Returns 0.0 for unsupported types — caller must verify TypeClass first.
Mirrors the dispatch in FB_TcOtelTaskTracer.AddAny so trace and metric
emission see numerics consistently.
*)
METHOD PRIVATE _AnyToLreal : LREAL
VAR_INPUT
    stArg : ANY;
END_VAR
VAR
    pBool  : POINTER TO BYTE;
    pSint  : POINTER TO SINT;
    pInt   : POINTER TO INT;
    pDint  : POINTER TO DINT;
    pLint  : POINTER TO LINT;
    pUsint : POINTER TO USINT;
    pUint  : POINTER TO UINT;
    pUdint : POINTER TO UDINT;
    pUlint : POINTER TO ULINT;
    pReal  : POINTER TO REAL;
    pLreal : POINTER TO LREAL;
END_VAR
CASE stArg.TypeClass OF
    __SYSTEM.TYPE_CLASS.TYPE_BOOL:
        pBool := stArg.pValue;
        IF pBool^ <> 0 THEN
            _AnyToLreal := 1.0;
        ELSE
            _AnyToLreal := 0.0;
        END_IF

    __SYSTEM.TYPE_CLASS.TYPE_SINT:
        pSint := stArg.pValue;
        _AnyToLreal := SINT_TO_LREAL(pSint^);

    __SYSTEM.TYPE_CLASS.TYPE_INT:
        pInt := stArg.pValue;
        _AnyToLreal := INT_TO_LREAL(pInt^);

    __SYSTEM.TYPE_CLASS.TYPE_DINT:
        pDint := stArg.pValue;
        _AnyToLreal := DINT_TO_LREAL(pDint^);

    __SYSTEM.TYPE_CLASS.TYPE_LINT:
        pLint := stArg.pValue;
        _AnyToLreal := LINT_TO_LREAL(pLint^);

    __SYSTEM.TYPE_CLASS.TYPE_USINT,
    __SYSTEM.TYPE_CLASS.TYPE_BYTE:
        pUsint := stArg.pValue;
        _AnyToLreal := USINT_TO_LREAL(pUsint^);

    __SYSTEM.TYPE_CLASS.TYPE_UINT,
    __SYSTEM.TYPE_CLASS.TYPE_WORD:
        pUint := stArg.pValue;
        _AnyToLreal := UINT_TO_LREAL(pUint^);

    __SYSTEM.TYPE_CLASS.TYPE_UDINT,
    __SYSTEM.TYPE_CLASS.TYPE_DWORD:
        pUdint := stArg.pValue;
        _AnyToLreal := UDINT_TO_LREAL(pUdint^);

    __SYSTEM.TYPE_CLASS.TYPE_ULINT,
    __SYSTEM.TYPE_CLASS.TYPE_LWORD:
        pUlint := stArg.pValue;
        _AnyToLreal := ULINT_TO_LREAL(pUlint^);

    __SYSTEM.TYPE_CLASS.TYPE_REAL:
        pReal := stArg.pValue;
        _AnyToLreal := REAL_TO_LREAL(pReal^);

    __SYSTEM.TYPE_CLASS.TYPE_LREAL:
        pLreal := stArg.pValue;
        _AnyToLreal := pLreal^;

    ELSE
        _AnyToLreal := 0.0;
END_CASE
END_METHOD

(*
:Description: Snapshot the current Welford aggregator into the body buffer.

Writes ``popcount(_nStatMask) * 8`` bytes — one LREAL per set bit, in
bit-index order (Min, Max, Mean, Sum, Count, StdDev). Returns FALSE on
body overflow without touching the buffer; the caller marks ``_bOverflow``.

Empty windows (no Observe call landed since the previous snapshot) still
produce a sample slot — all zeros — so ``sample_count`` keeps matching the
expected wall-clock cadence on the receiver side.
*)
METHOD PRIVATE _AppendAggregated : BOOL
VAR_INPUT
    (* Cycle offset for this sample relative to _nCycleStart. Only written
       when _bRecordSampleTimes is TRUE; ignored otherwise. Callers pass 0
       when they don't care. *)
    nCycleOff : UINT;
    (* Absolute DC time for this sample (raw F_GetActualDcTime64). Only
       written when _bRecordSampleTimesDc is TRUE; ignored otherwise. *)
    nDcSample : LINT;
END_VAR
VAR
    pDst    : POINTER TO BYTE;
    nOffset : UDINT;
    nStride : UDINT;
    fStdDev : LREAL;
    fCount  : LREAL;
END_VAR
nStride := _nSampleSize;
IF _bRecordSampleTimes THEN
    nStride := nStride + 2;
ELSIF _bRecordSampleTimesDc THEN
    nStride := nStride + 8;
END_IF
IF (_nBodyOffset + nStride) > BODY_CAPACITY THEN
    _AppendAggregated := FALSE;
    RETURN;
END_IF

pDst    := _ActiveBodyPtr() + _nBodyOffset;
IF _bRecordSampleTimes THEN
    Tc2_System.MEMCPY(pDst, ADR(nCycleOff), 2);
    pDst := pDst + 2;
ELSIF _bRecordSampleTimesDc THEN
    Tc2_System.MEMCPY(pDst, ADR(nDcSample), 8);
    pDst := pDst + 8;
END_IF
nOffset := 0;

IF (_nStatMask AND E_MetricStat.eMin) <> 0 THEN
    Tc2_System.MEMCPY(pDst + nOffset, ADR(_aggMin), 8);
    nOffset := nOffset + 8;
END_IF
IF (_nStatMask AND E_MetricStat.eMax) <> 0 THEN
    Tc2_System.MEMCPY(pDst + nOffset, ADR(_aggMax), 8);
    nOffset := nOffset + 8;
END_IF
IF (_nStatMask AND E_MetricStat.eMean) <> 0 THEN
    Tc2_System.MEMCPY(pDst + nOffset, ADR(_aggMean), 8);
    nOffset := nOffset + 8;
END_IF
IF (_nStatMask AND E_MetricStat.eSum) <> 0 THEN
    Tc2_System.MEMCPY(pDst + nOffset, ADR(_aggSum), 8);
    nOffset := nOffset + 8;
END_IF
IF (_nStatMask AND E_MetricStat.eCount) <> 0 THEN
    fCount := UDINT_TO_LREAL(_nAggCount);
    Tc2_System.MEMCPY(pDst + nOffset, ADR(fCount), 8);
    nOffset := nOffset + 8;
END_IF
IF (_nStatMask AND E_MetricStat.eStdDev) <> 0 THEN
    IF _nAggCount > 1 THEN
        fStdDev := SQRT(_aggSumSq / UDINT_TO_LREAL(_nAggCount - 1));
    ELSE
        fStdDev := 0.0;
    END_IF
    Tc2_System.MEMCPY(pDst + nOffset, ADR(fStdDev), 8);
    nOffset := nOffset + 8;
END_IF

_nBodyOffset      := _nBodyOffset + nStride;
_nSampleCount     := _nSampleCount + 1;
_AppendAggregated := TRUE;
END_METHOD

(*
:Description: Write one sample of the locked schema into the body buffer.

Returns FALSE when the body is full — caller sets ``_bOverflow``.
*)
METHOD PRIVATE _AppendSample : BOOL
VAR_INPUT
    stArg     : ANY;
    (* Cycle offset for this sample relative to _nCycleStart. Only written
       when _bRecordSampleTimes is TRUE; ignored otherwise. Callers pass 0
       when they don't care. *)
    nCycleOff : UINT;
    (* Absolute DC time for this sample (raw F_GetActualDcTime64). Only
       written when _bRecordSampleTimesDc is TRUE; ignored otherwise. *)
    nDcSample : LINT;
END_VAR
VAR
    fLreal     : LREAL;
    nStrLen    : UDINT;
    nCopyLen   : UDINT;
    nStride    : UDINT;
    pDst       : POINTER TO BYTE;
    pWstr      : POINTER TO WSTRING(255);
END_VAR
nStride := _nSampleSize;
IF _bRecordSampleTimes THEN
    nStride := nStride + 2;
ELSIF _bRecordSampleTimesDc THEN
    nStride := nStride + 8;
END_IF
IF (_nBodyOffset + nStride) > BODY_CAPACITY THEN
    _AppendSample := FALSE;
    RETURN;
END_IF

pDst := _ActiveBodyPtr() + _nBodyOffset;
IF _bRecordSampleTimes THEN
    Tc2_System.MEMCPY(pDst, ADR(nCycleOff), 2);
    pDst := pDst + 2;
ELSIF _bRecordSampleTimesDc THEN
    Tc2_System.MEMCPY(pDst, ADR(nDcSample), 8);
    pDst := pDst + 8;
END_IF

CASE _eBodySchema OF
    E_MetricBodySchema.eBool:
        IF Tc2_Utilities.PBYTE_TO_BYTE(stArg.pValue) <> 0 THEN
            pDst^ := 1;
        ELSE
            pDst^ := 0;
        END_IF

    E_MetricBodySchema.eNumeric:
        fLreal := _AnyToLreal(stArg);
        Tc2_System.MEMCPY(pDst, ADR(fLreal), 8);

    E_MetricBodySchema.eDiscrete:
        nCopyLen := DINT_TO_UDINT(stArg.diSize);
        IF nCopyLen > _nSampleSize THEN
            nCopyLen := _nSampleSize;
        END_IF
        Tc2_System.MEMCPY(pDst, stArg.pValue, nCopyLen);
        IF nCopyLen < _nSampleSize THEN
            Tc2_System.MEMSET(pDst + nCopyLen, 0, _nSampleSize - nCopyLen);
        END_IF

    E_MetricBodySchema.eString:
        Tc2_System.MEMSET(pDst, 0, _nSampleSize);
        nStrLen := Tc2_Utilities.LEN2(stArg.pValue);
        IF nStrLen > _nSampleSize THEN
            nStrLen := _nSampleSize;
        END_IF
        IF nStrLen > 0 THEN
            Tc2_System.MEMCPY(pDst, stArg.pValue, nStrLen);
        END_IF

    E_MetricBodySchema.eWstring:
        Tc2_System.MEMSET(pDst, 0, _nSampleSize);
        (* WLEN returns characters; we ship 2 B each, capped at _nSampleSize bytes.
           Typed-pointer cast first because WLEN can't take PVOID directly —
           same pattern FB_LogEntry._WriteWString uses. *)
        pWstr := stArg.pValue;
        nStrLen := INT_TO_UDINT(Tc2_Standard.WLEN(pWstr^)) * 2;
        IF nStrLen > _nSampleSize THEN
            nStrLen := _nSampleSize;
        END_IF
        IF nStrLen > 0 THEN
            Tc2_System.MEMCPY(pDst, stArg.pValue, nStrLen);
        END_IF

    ELSE
        _AppendSample := FALSE;
        RETURN;
END_CASE

_nBodyOffset  := _nBodyOffset + nStride;
_nSampleCount := _nSampleCount + 1;

_AppendSample := TRUE;
END_METHOD

(*
:Description: Flush if push window has elapsed.

Window timing is cycle-based (mirrors ``FB_TcOtelTaskDiag.CheckFlush``):
``target_cycles = push_interval_ms * 1000 / cycle_time_us``. Doesn't fire
when the buffer is empty — empty windows just slide the start cycle
forward.
*)
METHOD PRIVATE _CheckFlush
VAR
    nTaskIdx       : DINT;
    pTi            : POINTER TO PlcTaskSystemInfo;
    nNowCycle      : UDINT;
    nCycleTimeUs   : UDINT;
    nTargetCycles  : UDINT;
END_VAR
nTaskIdx := Tc2_Utilities.GETCURTASKINDEXEX();
IF nTaskIdx <= 0 THEN
    RETURN;
END_IF
pTi := ADR(TwinCAT_SystemInfoVarList._TaskInfo[nTaskIdx]);

nCycleTimeUs := pTi^.CycleTime / 10;
IF nCycleTimeUs = 0 THEN
    nCycleTimeUs := 1000; (* fallback: assume 1 ms *)
END_IF
nTargetCycles := (_nPushIntervalMs * 1000) / nCycleTimeUs;
IF nTargetCycles = 0 THEN
    nTargetCycles := 1;
END_IF

(* When per-sample timestamps are active, cap the window at the u16 ceiling
   so the per-sample cycle-offset never overflows. Observable effect: an
   earlier autoflush for extreme configs (e.g. 20 s push window on a 250 µs
   task). WithSpan pins may be consumed by the autoflush rather than the
   natural flush — use BindTracer for spans that outlive one window. *)
IF _bRecordSampleTimes AND nTargetCycles > 16#FFFF THEN
    nTargetCycles := 16#FFFF;
END_IF

nNowCycle := pTi^.CycleCount;
IF NOT _bWindowStartSet OR nNowCycle < _nWindowStartCycle THEN
    _nWindowStartCycle := nNowCycle;
    _bWindowStartSet   := TRUE;
    RETURN;
END_IF

IF (nNowCycle - _nWindowStartCycle) < nTargetCycles THEN
    RETURN;
END_IF

IF _nSampleCount > 0 THEN
    _DoFlush();
END_IF
_nWindowStartCycle := nNowCycle;
END_METHOD

(*
:Description: Finalize the active window into a sendable frame and enqueue for the sender.

Phase 8 — zero-copy queued dispatch:

1. If the previous window is still queued (``_bPending``) the sender has
   fallen behind. Increment ``_nDropWindow`` and reset the active half —
   we cannot touch the pending half nor duplicate ourselves in the queue.
2. Otherwise: build the header into a small stack staging (≤ ~160 B),
   MEMCPY the staged header into the active frame's reserve region so it
   sits directly before the body (one contiguous byte run), snapshot the
   pending metadata (buf index, hdr len, body len), flip ``_eActiveBuf``,
   reset the now-active (previously empty) half, and call
   ``sender.Enqueue(THIS)``.

The sender later calls ``_GetPendingPtr`` / ``_GetPendingLen`` to read the
frame pointer + length directly into ADSWRITE, and ``_NotifyFrameSent``
when the transfer completes. The body buffer is never MEMCPY'd.
*)
METHOD PRIVATE _DoFlush
VAR
    stHeader    : ST_PushMetricAggHeader;
    abyHdr      : ARRAY[0..255] OF BYTE;   // header(52) + trace(24) + name(63) + unit(15) + ns_len(1) + ns(127) ≤ 282
    nHdrLen     : UDINT;
    nNameLen    : UDINT;
    nUnitLen    : UDINT;
    nNsLen      : UDINT;
    byNsLen     : BYTE;
    refSender   : REFERENCE TO FB_TcOtelTaskMetrics;
    refSpan     : REFERENCE TO FB_Span;
    pActiveBase : POINTER TO BYTE;
END_VAR
(* Backlog guard: if the sender is still shipping our previous frame, the
   pending half is in use and we have no clean buffer to swap into. Drop
   this window rather than risk body corruption. In practice this only
   fires during a dead / slow tc-otel endpoint. *)
IF _bPending THEN
    _nDropWindow      := _nDropWindow + 1;
    _nBodyOffset      := 0;
    _nSampleCount     := 0;
    _bOverflow        := FALSE;
    _bWindowHasSample := FALSE;
    _nCycleStart      := 0;
    _nCycleEnd        := 0;
    _nDcTimeStart     := 0;
    _nDcTimeEnd       := 0;
    RETURN;
END_IF

(* Resolve trace context: per-flush WithSpan override beats persistent
   BindTracer. Both candidates and the chosen handle stay as REFERENCE TO —
   nullable via REF= 0 + __ISVALIDREF, no pointer round-trip needed. *)
refSpan REF= 0;
IF __ISVALIDREF(_pSpanOverride) THEN
    refSpan REF= _pSpanOverride;
ELSIF __ISVALIDREF(_pTracer) THEN
    refSpan REF= _pTracer.InnermostSpan;
END_IF

(* Build fixed header. *)
stHeader.nVersion         := 2;
stHeader.nEventType       := 21;
stHeader.nFlags           := 0;
IF _bOverflow THEN
    stHeader.nFlags := stHeader.nFlags OR 16#02;    (* bit1 = ring_overflowed *)
END_IF
IF __ISVALIDREF(refSpan) THEN
    stHeader.nFlags := stHeader.nFlags OR 16#01;    (* bit0 = has_trace_ctx *)
END_IF
IF _bRecordSampleTimes THEN
    stHeader.nFlags := stHeader.nFlags OR 16#04;    (* bit2 = has_sample_ts *)
END_IF
IF _bRecordSampleTimesDc THEN
    stHeader.nFlags := stHeader.nFlags OR 16#10;    (* bit4 = has_sample_ts_dc *)
END_IF
nNsLen := Tc2_Utilities.LEN2(ADR(_sLogger));
IF nNsLen > 127 THEN
    nNsLen := 127;
END_IF
IF nNsLen > 0 THEN
    stHeader.nFlags := stHeader.nFlags OR 16#08;    (* bit3 = has_namespace *)
END_IF
stHeader.eBodySchema      := _eBodySchema;
stHeader.nSampleSize      := _nSampleSize;
stHeader.nSampleCount     := _nSampleCount;
stHeader.nMetricId        := _nMetricId;
stHeader.nTaskIndex       := TO_USINT(Tc2_Utilities.GETCURTASKINDEXEX());
stHeader.nStatMask        := _nStatMask;
stHeader.nCycleCountStart := _nCycleStart;
stHeader.nCycleCountEnd   := _nCycleEnd;
stHeader.nDcTimeStart     := _nDcTimeStart;
stHeader.nDcTimeEnd       := _nDcTimeEnd;

nNameLen := Tc2_Utilities.LEN2(ADR(_sName));
IF nNameLen > 63 THEN
    nNameLen := 63;
END_IF
nUnitLen := Tc2_Utilities.LEN2(ADR(_sUnit));
IF nUnitLen > 15 THEN
    nUnitLen := 15;
END_IF
stHeader.nNameLen := TO_BYTE(nNameLen);
stHeader.nUnitLen := TO_BYTE(nUnitLen);

(* Stage [header | (trace_ctx) | name | unit] on the stack. *)
Tc2_System.MEMCPY(ADR(abyHdr), ADR(stHeader), SIZEOF(stHeader));
nHdrLen := SIZEOF(stHeader);

IF __ISVALIDREF(refSpan) THEN
    Tc2_System.MEMCPY(ADR(abyHdr) + nHdrLen,      ADR(refSpan._abTraceId[0]), 16);
    Tc2_System.MEMCPY(ADR(abyHdr) + nHdrLen + 16, ADR(refSpan._abSpanId[0]),  8);
    nHdrLen := nHdrLen + 24;
END_IF

(* Consume per-flush span override — BindTracer stays, WithSpan is one-shot. *)
_pSpanOverride REF= 0;

IF nNameLen > 0 THEN
    Tc2_System.MEMCPY(ADR(abyHdr) + nHdrLen, ADR(_sName), nNameLen);
    nHdrLen := nHdrLen + nNameLen;
END_IF
IF nUnitLen > 0 THEN
    Tc2_System.MEMCPY(ADR(abyHdr) + nHdrLen, ADR(_sUnit), nUnitLen);
    nHdrLen := nHdrLen + nUnitLen;
END_IF
IF nNsLen > 0 THEN
    (* Phase 2 scope-resolver: ns_len(1) + namespace(ns_len). *)
    byNsLen := TO_BYTE(nNsLen);
    Tc2_System.MEMCPY(ADR(abyHdr) + nHdrLen,     ADR(byNsLen),   1);
    Tc2_System.MEMCPY(ADR(abyHdr) + nHdrLen + 1, ADR(_sLogger),  nNsLen);
    nHdrLen := nHdrLen + 1 + nNsLen;
END_IF

(* Defensive clamp: the header reserve is HDR_RESERVE bytes. Oversized
   headers would overlap the body. In practice nHdrLen ≤ 154. *)
IF nHdrLen > HDR_RESERVE THEN
    _nDropEmit := _nDropEmit + 1;
    (* Reset window and bail — don't corrupt the frame layout. *)
    _nBodyOffset      := 0;
    _nSampleCount     := 0;
    _bOverflow        := FALSE;
    _bWindowHasSample := FALSE;
    _nCycleStart      := 0;
    _nCycleEnd        := 0;
    _nDcTimeStart     := 0;
    _nDcTimeEnd       := 0;
    RETURN;
END_IF

(* Position the staged header so its last byte sits at offset HDR_RESERVE-1
   of the active frame — i.e. flush against the body start. Single MEMCPY
   of ≤ 160 B; no body copy. *)
pActiveBase := _ActiveFrameAddr();
Tc2_System.MEMCPY(pActiveBase + (HDR_RESERVE - nHdrLen), ADR(abyHdr), nHdrLen);

(* Snapshot pending metadata: the active (now-to-be-shipped) half. *)
_ePendingBuf     := _eActiveBuf;
_nPendingHdrLen  := nHdrLen;
_nPendingBodyLen := _nBodyOffset;
_bPending        := TRUE;

(* Flip active → the other half. Reset the new-active mutable state. *)
IF _eActiveBuf = 0 THEN
    _eActiveBuf := 1;
ELSE
    _eActiveBuf := 0;
END_IF
_nBodyOffset      := 0;
_nSampleCount     := 0;
_bOverflow        := FALSE;
_bWindowHasSample := FALSE;
_nCycleStart      := 0;
_nCycleEnd        := 0;
_nDcTimeStart     := 0;
_nDcTimeEnd       := 0;

(* Hand the pending half to the sender's dispatch ring. *)
refSender REF= PRG_TaskLog.TaskMetrics;
IF __ISVALIDREF(refSender) THEN
    IF NOT refSender.Enqueue(THIS) THEN
        (* Ring overflow — real drop. Release the pending half so the next
           window can still flush, and count as emit drop. *)
        _bPending  := FALSE;
        _nDropEmit := _nDropEmit + 1;
    END_IF
ELSE
    (* Sender missing — treat like ring overflow. *)
    _bPending  := FALSE;
    _nDropEmit := _nDropEmit + 1;
END_IF
END_METHOD

(*
:Description: INTERNAL — total bytes of the frame currently in the sender queue.

Called by ``FB_TcOtelTaskMetrics._KickHead`` to populate ADSWRITE.LEN.
Returns 0 when ``_bPending`` is FALSE (spurious call — sender should ignore).
*)
METHOD INTERNAL _GetPendingLen : UDINT
IF _bPending THEN
    _GetPendingLen := _nPendingHdrLen + _nPendingBodyLen;
ELSE
    _GetPendingLen := 0;
END_IF
END_METHOD

(*
:Description: INTERNAL — byte pointer to the first byte of the pending frame.

Frame layout in the pending half (``_ePendingBuf``):
  [HDR_RESERVE - _nPendingHdrLen .. HDR_RESERVE - 1]  header + trace + name + unit
  [HDR_RESERVE .. HDR_RESERVE + _nPendingBodyLen - 1] body samples
So the frame starts at ``frame[HDR_RESERVE - _nPendingHdrLen]`` and runs
``_nPendingHdrLen + _nPendingBodyLen`` bytes — a single contiguous ADS range.

Called by ``FB_TcOtelTaskMetrics._KickHead`` to populate ADSWRITE.SRCADDR.
Returns 0 when no frame is pending.
*)
METHOD INTERNAL _GetPendingPtr : PVOID
IF NOT _bPending THEN
    _GetPendingPtr := 0;
    RETURN;
END_IF

IF _ePendingBuf = 0 THEN
    _GetPendingPtr := ADR(_aFrameA[0]) + (HDR_RESERVE - _nPendingHdrLen);
ELSE
    _GetPendingPtr := ADR(_aFrameB[0]) + (HDR_RESERVE - _nPendingHdrLen);
END_IF
END_METHOD

(*
:Description: Map the IEC type class of the first Observe call to a body schema.

Returns FALSE for unsupported types (TIME, DATE, structures, arrays, etc.)
so Observe can drop those gracefully and surface via _nWrongTypeDrops.
*)
METHOD PRIVATE _LockSchema : BOOL
VAR_INPUT
    stArg : ANY;
END_VAR
CASE stArg.TypeClass OF
    __SYSTEM.TYPE_CLASS.TYPE_BOOL:
        _eBodySchema := E_MetricBodySchema.eBool;
        _nSampleSize := 1;

    __SYSTEM.TYPE_CLASS.TYPE_SINT,
    __SYSTEM.TYPE_CLASS.TYPE_INT,
    __SYSTEM.TYPE_CLASS.TYPE_DINT,
    __SYSTEM.TYPE_CLASS.TYPE_LINT,
    __SYSTEM.TYPE_CLASS.TYPE_USINT,
    __SYSTEM.TYPE_CLASS.TYPE_UINT,
    __SYSTEM.TYPE_CLASS.TYPE_UDINT,
    __SYSTEM.TYPE_CLASS.TYPE_ULINT,
    __SYSTEM.TYPE_CLASS.TYPE_REAL,
    __SYSTEM.TYPE_CLASS.TYPE_LREAL:
        IF _nStatMask <> 0 THEN
            _eBodySchema := E_MetricBodySchema.eNumericAggregated;
            _nSampleSize := _nAggSampleSize;
        ELSE
            _eBodySchema := E_MetricBodySchema.eNumeric;
            _nSampleSize := 8;     (* widened to LREAL *)
        END_IF

    __SYSTEM.TYPE_CLASS.TYPE_BYTE,
    __SYSTEM.TYPE_CLASS.TYPE_WORD,
    __SYSTEM.TYPE_CLASS.TYPE_DWORD,
    __SYSTEM.TYPE_CLASS.TYPE_LWORD,
    __SYSTEM.TYPE_CLASS.TYPE_ENUM:
        _eBodySchema := E_MetricBodySchema.eDiscrete;
        _nSampleSize := DINT_TO_UDINT(stArg.diSize);

    __SYSTEM.TYPE_CLASS.TYPE_STRING:
        _eBodySchema := E_MetricBodySchema.eString;
        _nSampleSize := _nStringSize;
        F_InternalLog(
            E_LogLevel.eWarn,
            'FB_Metrics._LockSchema',
            'Unsupported TypeClass=%d for metric %s',
            Tc2_Utilities.F_UDINT(stArg.TypeClass),
            Tc2_Utilities.F_StringEx(_sName),
            Tc2_Utilities.EMPTY_ARG_VALUE,
            Tc2_Utilities.EMPTY_ARG_VALUE
        );
        _LockSchema := FALSE;
        RETURN;

    __SYSTEM.TYPE_CLASS.TYPE_WSTRING:
        _eBodySchema := E_MetricBodySchema.eWstring;
        _nSampleSize := _nStringSize * 2;
        F_InternalLog(
            E_LogLevel.eWarn,
            'FB_Metrics._LockSchema',
            'Unsupported TypeClass=%d for metric %s',
            Tc2_Utilities.F_UDINT(stArg.TypeClass),
            Tc2_Utilities.F_StringEx(_sName),
            Tc2_Utilities.EMPTY_ARG_VALUE,
            Tc2_Utilities.EMPTY_ARG_VALUE
        );
        _LockSchema := FALSE;
        RETURN;

    ELSE
        F_InternalLog(
            E_LogLevel.eWarn,
            'FB_Metrics._LockSchema',
            'Unsupported TypeClass=%d for metric %s',
            Tc2_Utilities.F_UDINT(stArg.TypeClass),
            Tc2_Utilities.F_StringEx(_sName),
            Tc2_Utilities.EMPTY_ARG_VALUE,
            Tc2_Utilities.EMPTY_ARG_VALUE
        );
        _LockSchema := FALSE;
        RETURN;
END_CASE

_nLockedTypeClass := stArg.TypeClass;
_LockSchema       := TRUE;
END_METHOD

(*
:Description: INTERNAL — sender completion callback.

Called by ``FB_TcOtelTaskMetrics.Call`` once ADSWRITE finishes (success, ADS
error, or watchdog). Releases the pending half so the next ``_DoFlush`` can
swap into it, and updates per-metric counters.

Do not call from user code.
*)
METHOD INTERNAL _NotifyFrameSent
VAR_INPUT
    bOk : BOOL;
END_VAR
IF bOk THEN
    _nFlushOk := _nFlushOk + 1;
ELSE
    _nDropEmit := _nDropEmit + 1;
END_IF

_bPending        := FALSE;
_nPendingHdrLen  := 0;
_nPendingBodyLen := 0;
END_METHOD

(*
:Description: Live DC time, falling back to cycle-start task DC time.

Same fallback as FB_TcOtelTaskTracer._NowDcTime — keeps metric and trace
timestamps comparable.
*)
METHOD PRIVATE _NowDcTime : LINT
VAR
    nTaskIdx : DINT;
END_VAR
_NowDcTime := TO_LINT(Tc2_EtherCAT.F_GetActualDcTime64());
IF _NowDcTime = 0 THEN
    nTaskIdx := Tc2_Utilities.GETCURTASKINDEXEX();
    IF nTaskIdx > 0 THEN
        _NowDcTime := TwinCAT_SystemInfoVarList._TaskInfo[nTaskIdx].DcTaskTime;
    END_IF
END_IF
END_METHOD

(*
:Description: Bit-count of a BYTE — used to size the aggregated sample.

Trivial loop is fine for an 8-bit value; called once per SetAggregation,
not per cycle.
*)
METHOD PRIVATE _PopCount8 : UDINT
VAR_INPUT
    nByte : BYTE;
END_VAR
VAR
    nBit : INT;
END_VAR
_PopCount8 := 0;
FOR nBit := 0 TO 7 DO
    IF (nByte AND SHL(BYTE#1, nBit)) <> 0 THEN
        _PopCount8 := _PopCount8 + 1;
    END_IF
END_FOR
END_METHOD

(*
:Description: Bind this metric to an FB_TcOtelTracer for trace exemplar correlation.

Read-at-flush-time semantic: every ``_DoFlush`` snapshots the tracer's
**currently** innermost-open span (trace_id + span_id) into the wire
header. The span's ID gets promoted to an OTel Exemplar on every data
point in that batch so Grafana / Tempo render "View trace" links.

What ends up on the frame:

* a span is open on the bound tracer at flush time → that span's trace_id
* no span open (all ``End``'d, or never ``Begin``'d) → no trace bytes, frame is 24 B shorter
* ``BindTracer(0)`` → no trace bytes

A span that opens **and** closes between two flushes leaves no trace on
either frame — if that matters, use ``WithSpan`` or call ``Flush``
before ``End``.

Pass ``0`` to unbind. Idempotent — safe to call repeatedly.

**Example**

.. code-block:: pascal

    VAR
        _tracer : FB_TcOtelTracer;
        _temp   : FB_Metrics;
    END_VAR

    IF _TaskInfo[GETCURTASKINDEXEX()].FirstCycle THEN
        _temp.Init('motor.temperature', 'celsius');
        _temp.BindTracer(_tracer);
    END_IF
*)
METHOD PUBLIC BindTracer : BOOL
VAR_INPUT
    pTracer : REFERENCE TO FB_Trace;
END_VAR
_pTracer REF= pTracer;
BindTracer := TRUE;
END_METHOD

(*
:Description: Drives push-window check.

Only needed when the user calls ``Observe`` sporadically (so a long quiet
period would otherwise delay flush past its window). When ``Observe`` is
called every cycle this is redundant but harmless.
*)
METHOD PUBLIC Call
IF _bInitialized THEN
    _CheckFlush();
END_IF
END_METHOD

(*
:Description: Flush any buffered samples before this FB instance is destroyed.

Online change / program stop / FB deletion all route through here — without
this, the last partial window would be silently lost.
*)
METHOD FB_exit : BOOL
VAR_INPUT
    bInCopyCode : BOOL;
END_VAR
(* Cold Reset / RT shutdown destroys FB instances in undefined order.
   PRG_TaskLog.TaskMetrics may be torn down before us; calling
   Dequeue on a dangling reference segfaults inside the AuxTask
   (__ISVALIDREF catches NULL only, not dangling-after-free). Buffered
   samples on shutdown are lost — acceptable, no consumer remains
   after the Reset.

   Online change (bInCopyCode = TRUE) preserves both old and new
   instances in memory; flushing here would double-emit if the new
   instance also flushes. *)
FB_exit := TRUE;
END_METHOD

// Phase 2 scope-resolver: derive _sLogger from the FB's instance
// path. Strips library + application + variable-name segments,
// leaving (e.g.) ``PRG_TestSimpleApi.fbMotor`` so the OTel
// ScopeResolver maps the frame to the OWNING FB's type for
// ``InstrumentationScope.name``. Mirrors FB_Log.FB_Init.
METHOD FB_Init: BOOL
VAR_INPUT
    bInitRetains: BOOL;
    bInCopyCode: BOOL;
END_VAR
VAR
    nFindIdx : INT;
    i        : INT;
    nLastDot : INT;
END_VAR
nFindIdx := Tc2_Standard.FIND(_sInstancePath, '.');
IF nFindIdx > 0 THEN
    _sInstancePath := Tc2_Standard.DELETE(_sInstancePath, nFindIdx + 1, 0);
    nFindIdx := Tc2_Standard.FIND(_sInstancePath, '.');
    IF nFindIdx > 0 THEN
        _sInstancePath := Tc2_Standard.DELETE(_sInstancePath, nFindIdx + 1, 0);
        nLastDot := 0;
        FOR i := Tc2_Standard.LEN(_sInstancePath) TO 1 BY -1 DO
            IF Tc2_Standard.MID(_sInstancePath, 1, i) = '.' THEN
                nLastDot := i;
                EXIT;
            END_IF
        END_FOR
        IF nLastDot > 1 THEN
            _sLogger := Tc2_Standard.LEFT(_sInstancePath, nLastDot - 1);
        ELSE
            _sLogger := _sInstancePath;
        END_IF
    END_IF
END_IF

FB_Init := TRUE;
END_METHOD

(*
:Description: Force-flush the buffered samples now, regardless of push window.

No-op when the buffer is empty.
*)
METHOD PUBLIC Flush : BOOL
IF _bInitialized AND _nSampleCount > 0 THEN
    _DoFlush();
END_IF
Flush := TRUE;
END_METHOD

(*
:Description: One-time configuration of the metric identity.

Idempotent — recomputes the FNV-1a metric id from the current name. Safe
to call from FirstCycle. ``nStringSize`` is only meaningful when the
locked schema turns out to be eString / eWstring; ignored for numerics.
*)
METHOD PUBLIC Init : BOOL
VAR_INPUT
    sName       : STRING(63);
    sUnit       : STRING(15) := '';
    nStringSize : UDINT      := 64;       // bytes per string sample (chars for WSTRING)
END_VAR
VAR
    i      : INT;
    nLen   : INT;
    nHash  : UDINT;
    pBytes : POINTER TO BYTE;
END_VAR
_sName       := sName;
_sUnit       := sUnit;
_nStringSize := nStringSize;
IF _nStringSize = 0 THEN
    _nStringSize := 64;
END_IF
IF _nStringSize > 255 THEN
    _nStringSize := 255;
END_IF

(* FNV-1a 32-bit over the name bytes. Stable across runs as long as the
   name string doesn't change. *)
nHash := UDINT#16#811C9DC5;
nLen  := Tc2_Standard.LEN(_sName);
IF nLen > 0 THEN
    pBytes := ADR(_sName);
    FOR i := 0 TO nLen - 1 DO
        nHash := (nHash XOR BYTE_TO_UDINT(pBytes[i])) * UDINT#16#01000193;
    END_FOR
END_IF
_nMetricId    := nHash;

_bInitialized := TRUE;
Init          := TRUE;
END_METHOD

PROPERTY PUBLIC MetricId : UDINT
GET
MetricId := _nMetricId;
END_GET
END_PROPERTY

(*
:Description: Capture one observation of the metric value.

Returns FALSE only on hard errors (Init not called, unsupported type on
first call, type changed after lock). Successful sample-suppression by
rate-limit or change-detect still returns TRUE — the FB did its job by
deciding the value didn't need to be stored.

Safe to call every cycle — internal rate-limit makes that cheap.
*)
METHOD PUBLIC Observe : BOOL
VAR_INPUT
    stArg : ANY;
END_VAR
VAR
    nTaskIdx       : DINT;
    pTi            : POINTER TO PlcTaskSystemInfo;
    nNowCycle      : UDINT;
    nCycleTimeUs   : UDINT;
    nSampleTargetCycles : UDINT;
    nCmpLen        : UDINT;
    nDcNow         : LINT;
    fLrealForAgg   : LREAL;     // widened sample for the online aggregator
    bAggMode       : BOOL;      // shorthand for "stat-mask aggregation active"
    nCycleOff      : UINT;      // per-sample offset for optional sample-TS
END_VAR
IF NOT _bInitialized OR stArg.pValue = 0 THEN
    Observe := FALSE;
    RETURN;
END_IF

IF _eBodySchema = E_MetricBodySchema.eString OR _eBodySchema = E_MetricBodySchema.eWstring THEN
	_nWrongTypeDrops := _nWrongTypeDrops + 1;
	Observe := FALSE;
	RETURN;
END_IF

(* Lock schema on first call. *)
IF _eBodySchema = E_MetricBodySchema.eUnknown THEN
    IF NOT _LockSchema(stArg) THEN
        _nWrongTypeDrops := _nWrongTypeDrops + 1;
        Observe := FALSE;
        RETURN;
    END_IF
ELSIF _nLockedTypeClass <> stArg.TypeClass THEN
    F_InternalLog(
        E_LogLevel.eWarn,
        'FB_Metrics.Observe',
        'TypeClass mismatch for %s (locked=%d got=%d)',
        Tc2_Utilities.F_StringEx(_sName),
        Tc2_Utilities.F_UDINT(_nLockedTypeClass),
        Tc2_Utilities.F_UDINT(stArg.TypeClass),
        Tc2_Utilities.EMPTY_ARG_VALUE
    );
    _nWrongTypeDrops := _nWrongTypeDrops + 1;
    Observe := FALSE;
    RETURN;
END_IF

nTaskIdx := Tc2_Utilities.GETCURTASKINDEXEX();
IF nTaskIdx <= 0 THEN
    Observe := FALSE;
    RETURN;
END_IF
pTi := ADR(TwinCAT_SystemInfoVarList._TaskInfo[nTaskIdx]);
nNowCycle := pTi^.CycleCount;

bAggMode := _eBodySchema = E_MetricBodySchema.eNumericAggregated;

(* Aggregation: in eNumericAggregated mode the aggregator absorbs every
   single Observe call (Welford online for mean/stddev). The rate-limit
   below still gates how often we *snapshot* the aggregator into the body
   buffer — but no value is dropped between ticks. *)
IF bAggMode THEN
    fLrealForAgg := _AnyToLreal(stArg);
    _AggUpdate(fLrealForAgg);
END_IF

(* Sample-interval rate limit (cycle-based, derived from CycleTime). *)
IF _nSampleIntervalMs > 0 AND _bLastSampleSet THEN
    nCycleTimeUs := pTi^.CycleTime / 10;
    IF nCycleTimeUs = 0 THEN
        nCycleTimeUs := 1000;
    END_IF
    nSampleTargetCycles := (_nSampleIntervalMs * 1000) / nCycleTimeUs;
    IF nSampleTargetCycles = 0 THEN
        nSampleTargetCycles := 1;
    END_IF
    IF (nNowCycle - _nLastSampleCycle) < nSampleTargetCycles THEN
        Observe := TRUE;
        RETURN;
    END_IF
END_IF

(* Change-detect path (raw mode only — for aggregated mode every Observe
   already updated the aggregator above, no point in suppressing). *)
IF NOT bAggMode AND _bChangeDetect AND _bLastValueValid THEN
    nCmpLen := _nSampleSize;
    IF nCmpLen > SIZEOF(_abyLastValue) THEN
        nCmpLen := SIZEOF(_abyLastValue);
    END_IF
    IF Tc2_System.MEMCMP(stArg.pValue, ADR(_abyLastValue), nCmpLen) = 0 THEN
        (* Even on no-change we still update last-sample timestamp so the
           rate-limit window resets — so a value that resumes changing right
           after the interval doesn't have to wait an extra slot. *)
        _nLastSampleCycle := nNowCycle;
        _bLastSampleSet   := TRUE;
        Observe := TRUE;
        RETURN;
    END_IF
END_IF

(* Window timing must be established BEFORE the append so the per-sample
   cycle offset is well-defined on the very first sample. Moving this block
   up changes no observable semantics in the default path — _nCycleStart /
   _nDcTimeStart were overwritten by this sample anyway — but guarantees
   that _bRecordSampleTimes sees a valid reference point. *)
nDcNow := _NowDcTime();
IF NOT _bWindowHasSample THEN
    _nCycleStart      := nNowCycle;
    _nDcTimeStart     := nDcNow;
    _bWindowHasSample := TRUE;
END_IF
_nCycleEnd   := nNowCycle;
_nDcTimeEnd  := nDcNow;

(* u16 offset: safe because _CheckFlush caps the window at 0xFFFF cycles
   whenever _bRecordSampleTimes is active. When the flag is off, the value
   is unused but we still clamp defensively. *)
IF (nNowCycle - _nCycleStart) > 16#FFFF THEN
    nCycleOff := 16#FFFF;
ELSE
    nCycleOff := TO_UINT(nNowCycle - _nCycleStart);
END_IF

IF bAggMode THEN
    (* Snapshot the aggregator into the body, then reset for the next window.
       _AppendAggregated falls through to FALSE only on body overflow — bail
       early in that case, the old aggregator state would be wrong to keep
       around for the next snapshot anyway. *)
    IF NOT _AppendAggregated(nCycleOff, nDcNow) THEN
        _bOverflow   := TRUE;
        _nDropAppend := _nDropAppend + 1;
    END_IF
    _AggReset();
ELSE
    (* Raw append (single value per sample tick). *)
    IF NOT _AppendSample(stArg, nCycleOff, nDcNow) THEN
        _bOverflow   := TRUE;
        _nDropAppend := _nDropAppend + 1;
    END_IF

    (* Update last-value cache regardless of append success — change-detect
       should still suppress the next no-change observation. *)
    nCmpLen := _nSampleSize;
    IF nCmpLen > SIZEOF(_abyLastValue) THEN
        nCmpLen := SIZEOF(_abyLastValue);
    END_IF
    Tc2_System.MEMCPY(ADR(_abyLastValue), stArg.pValue, nCmpLen);
    _bLastValueValid := TRUE;
END_IF

_nLastSampleCycle := nNowCycle;
_bLastSampleSet   := TRUE;

(* Mid-window autoflush: when the body crosses the high-water mark we
   swap halves immediately rather than wait for _CheckFlush's push-
   interval tick. Keeps oversampling bursts streaming when one push
   window otherwise wouldn't fit.

   Critical guard — only fire when the pending half is FREE. If the
   sender is still shipping the previous frame, _DoFlush would see
   _bPending=TRUE, reset the entire active half to empty, and bump
   _nDropWindow — throwing away every sample we accumulated in the
   burst. That makes the case autoflush was designed for strictly
   worse than just letting the body hit 100 % and dropping one
   sample at a time via _nDropAppend. So: when pending is busy we
   hold off and keep filling. If we reach 100 % before pending
   drains, _AppendSample returns FALSE and we lose one sample — not
   the whole window. *)
IF _nBodyOffset >= BODY_HIGH_WATER AND NOT _bPending THEN
    _DoFlush();
END_IF

_CheckFlush();

Observe := TRUE;
END_METHOD

PROPERTY PUBLIC SampleCount : UDINT
GET
SampleCount := _nSampleCount;
END_GET
END_PROPERTY

(*
:Description: Enable / change online aggregation over the sample interval.

``nMask`` is a bitmask **OR-combined from individual ``E_MetricStat``
values**. Each set bit selects one statistic to compute via Welford
online aggregation and ship per sample tick:

==================== === ===============================================
Bit                  Hex Stat shipped per sample
==================== === ===============================================
``E_MetricStat.eMin``    1   minimum observed value
``E_MetricStat.eMax``    2   maximum observed value
``E_MetricStat.eMean``   4   arithmetic mean
``E_MetricStat.eSum``    8   sum (totalizer — energy, parts, distance)
``E_MetricStat.eCount`` 16   observations folded (gap / drop detection)
``E_MetricStat.eStdDev`` 32   standard deviation (jitter / stability)
==================== === ===============================================

The bits ship in **bit-index order** (Min first if set, then Max, Mean,
Sum, Count, StdDev). Wire size per sample = ``popcount(nMask) * 8``.

.. code-block:: pascal

	// Raw - use raw value (last), 8 B/sample (Default)
	fbEnergy.SetAggregation(0);

    // Counter — totalizer only, 8 B/sample.
    fbEnergy.SetAggregation(E_MetricStat.eSum);

    // Envelope — min + max, 16 B/sample. Catch peaks/troughs.
    fbTemp.SetAggregation(E_MetricStat.eMin OR E_MetricStat.eMax);

    // Standard — min + max + mean, 24 B/sample. Recommended default.
    fbProcess.SetAggregation(
        E_MetricStat.eMin OR E_MetricStat.eMax OR E_MetricStat.eMean);

    // Full — all six, 48 B/sample. Diagnostic / tuning.
    fbCritical.SetAggregation(
        E_MetricStat.eMin OR E_MetricStat.eMax OR E_MetricStat.eMean
        OR E_MetricStat.eSum OR E_MetricStat.eCount OR E_MetricStat.eStdDev);

Pass ``0`` to revert to raw single-value sampling. With aggregation
enabled, every ``Observe`` call updates the Welford aggregator
regardless of rate-limit; the rate-limit then controls how often the
aggregator is *snapshotted* into the body buffer. So values that
appear between sample ticks are no longer dropped — they're folded
into the next snapshot's min/max/mean/etc.

Aggregation is numeric-only. On non-numeric metrics (BOOL, STRING,
WSTRING, ENUM/discrete) the mask is ignored and a warning is logged
the first time. The mask is a hint applied at the next ``Observe``;
in-flight body content is not retroactively converted, so call
``SetAggregation`` at startup before the first ``Observe``.
*)
METHOD PUBLIC SetAggregation : BOOL
VAR_INPUT
    nMask : BYTE;
END_VAR
_nStatMask      := nMask;
_nAggSampleSize := _PopCount8(nMask) * 8;

(* If the schema is already locked to a numeric type, switch in/out of
   the aggregated body schema on the fly so the next sample tick uses
   the right write path. For non-numeric locked types the mask is held
   but never consumed (the locked schema decides which append-path runs);
   warn once so the user knows it's a no-op. *)
IF _eBodySchema = E_MetricBodySchema.eNumeric AND nMask <> 0 THEN
    _eBodySchema := E_MetricBodySchema.eNumericAggregated;
    _nSampleSize := _nAggSampleSize;
ELSIF _eBodySchema = E_MetricBodySchema.eNumericAggregated AND nMask = 0 THEN
    _eBodySchema := E_MetricBodySchema.eNumeric;
    _nSampleSize := 8;
ELSIF _eBodySchema = E_MetricBodySchema.eNumericAggregated AND nMask <> 0 THEN
    _nSampleSize := _nAggSampleSize;
ELSIF nMask <> 0 AND (_eBodySchema = E_MetricBodySchema.eBool
                   OR _eBodySchema = E_MetricBodySchema.eString
                   OR _eBodySchema = E_MetricBodySchema.eWstring
                   OR _eBodySchema = E_MetricBodySchema.eDiscrete) THEN
    F_InternalLog(
        E_LogLevel.eWarn,
        'FB_Metrics.SetAggregation',
        'Aggregation only valid for numeric metrics — %s is non-numeric, mask ignored',
        Tc2_Utilities.F_StringEx(_sName),
        Tc2_Utilities.EMPTY_ARG_VALUE,
        Tc2_Utilities.EMPTY_ARG_VALUE,
        Tc2_Utilities.EMPTY_ARG_VALUE
    );
END_IF

_AggReset();
SetAggregation := TRUE;
END_METHOD

(*
:Description: Enable / disable byte-wise change-detect (default TRUE).

Disable when you want to capture every cycle's value as-is even if it
hasn't changed (e.g. for "still alive" continuity at slow sample rates).
*)
METHOD PUBLIC SetChangeDetect : BOOL
VAR_INPUT
    bEnabled : BOOL;
END_VAR
_bChangeDetect := bEnabled;
SetChangeDetect := TRUE;
END_METHOD

(*
:Description: How often to flush the buffer to tc-otel (default 1000 ms).

Lower bound is one task cycle. Smaller values mean more frames on the wire;
larger values risk buffer overflow on high-rate metrics (8 KB ÷ sample_size).
*)
METHOD PUBLIC SetPushIntervalMs : BOOL
VAR_INPUT
    nMs : UDINT;
END_VAR
_nPushIntervalMs := nMs;
IF _nPushIntervalMs = 0 THEN
    _nPushIntervalMs := 1000;
END_IF
SetPushIntervalMs := TRUE;
END_METHOD

(*
:Description: Enable / disable per-sample timestamp emission (default FALSE).

When TRUE every body slot is prefixed with a 2-byte little-endian u16 cycle
offset relative to ``cycle_count_start``, and the wire header carries
``flags.bit2 = METRIC_FLAG_HAS_SAMPLE_TS``. Receivers use the offset to
reconstruct accurate per-sample DC times instead of linearly interpolating
across the window.

Use this when sampling is irregular — change-detect bursts, sporadic
``Observe`` calls, or `SetSampleIntervalMs` rate-limiting in combination with
bursty input. When ``Observe`` runs every task cycle, default linear
interpolation is already exact and this opt-in costs 2 B per sample for
nothing.

Side effects:

* ``_CheckFlush`` caps the push window at ``0xFFFF`` task cycles whenever
  this flag is active. On a 250 µs task that is ~16 s; on a 1 ms task
  ~65 s — well beyond any realistic metric interval. Configurations that
  would exceed the cap are silently autoflushed earlier.
* ``WithSpan`` overrides are one-shot and get consumed by the *next* flush,
  which may now be an autoflush rather than the natural window end. For
  spans that outlive one window, prefer ``BindTracer``.
* ``SetAggregation`` splits the Welford state across autoflushes, which
  produces finer-grained stat windows downstream. Acceptable for most
  dashboards; note if you rely on exact per-window moments.

Cost per sample when active: 2 B prefix. Bool (1 B) body grows to 3 B,
Numeric (8 B) to 10 B, NumericAggregated with full stat mask (48 B) to
50 B. Zero overhead when disabled.
*)
METHOD PUBLIC SetRecordSampleTimes : BOOL
VAR_INPUT
    bEnable : BOOL;
END_VAR
_bRecordSampleTimes := bEnable;
IF bEnable THEN
    (* The two sample-ts modes are mutually exclusive — the wire format
       carries them in separate flag bits but only one prefix layout per
       slot. Turning u16-offset mode on forces DC-mode off. *)
    _bRecordSampleTimesDc := FALSE;
END_IF
SetRecordSampleTimes := TRUE;
END_METHOD

(*
:Description: Enable / disable per-sample i64 absolute DC time emission (default FALSE).

Use this for **true oversampling** — when `Observe` is called more than once
per task cycle and every observation must reach the backend as its own
distinct datapoint. The u16-offset mode (``SetRecordSampleTimes``) collapses
all same-cycle samples onto one offset value; this mode emits the raw
``F_GetActualDcTime64()`` reading instead so the receiver can resolve them.

When TRUE every body slot is prefixed with an 8-byte little-endian i64
absolute DC time, and the wire header carries
``flags.bit4 = METRIC_FLAG_HAS_SAMPLE_TS_DC (0x10)``. The receiver uses
``dc_time[i]`` directly as the per-sample timestamp — no interpolation,
no dependency on ``cycle_count_*``.

**Honest timestamps, no synthetic tiebreaker**: if two consecutive
``Observe`` calls inside one task cycle happen faster than the hardware
DC clock ticks, the emitted DC times can be identical. Those duplicates
are real and may be deduplicated by storage backends with last-value-
wins semantics on identical timestamps. The PLC deliberately does *not*
fabricate a fake monotonic increment because that would lie about when
the observation actually happened.

**Mutually exclusive with ``SetRecordSampleTimes``** — calling
``SetRecordSampleTimesDc(TRUE)`` while u16-offset mode is on forces
u16-offset off, and vice versa.

**Cost** per sample when active: 8 B prefix. Bool (1 B) body grows to
9 B, Numeric (8 B) to 16 B, NumericAggregated with full stat mask
(48 B) to 56 B. Zero overhead when disabled.

**Buffer impact**: with 16 B Numeric stride the 32 KB body holds ~2048
samples per half before mid-window autoflush kicks in (at the 80 %
high-water mark). Pair with a push interval ≤ 200 ms for sustained
oversampling so the sender keeps draining between bursts.
*)
METHOD PUBLIC SetRecordSampleTimesDc : BOOL
VAR_INPUT
    bEnable : BOOL;
END_VAR
_bRecordSampleTimesDc := bEnable;
IF bEnable THEN
    _bRecordSampleTimes := FALSE;
END_IF
SetRecordSampleTimesDc := TRUE;
END_METHOD

(*
:Description: Minimum interval between captured samples (default 0 = every change).

Set > 0 to rate-limit a fast-changing value: at most one sample per ``nMs``
ms reaches the buffer, regardless of how often Observe is called.
*)
METHOD PUBLIC SetSampleIntervalMs : BOOL
VAR_INPUT
    nMs : UDINT;
END_VAR
_nSampleIntervalMs := nMs;
SetSampleIntervalMs := TRUE;
END_METHOD

(*
:Description: Override the trace-context snapshot for the very next flush.

One-shot — consumed by ``_DoFlush`` and cleared. Subsequent flushes fall
back to the ``BindTracer``-bound innermost span, or no trace at all if
neither is set.

Unlike ``BindTracer``, ``WithSpan`` captures the span **immediately**,
so it still pins the correct trace_id even if the span is ``End``'d
before flush actually runs. This is the correct tool when:

* a short-lived span closes inside the push window and you want the
  window's metrics tagged with its ID, or
* you want a specific span tagged instead of whichever happens to be
  innermost at flush time.

Typical pattern for "this metric window belongs to span X":

.. code-block:: pascal

    _spn.Begin('quick_op');
    _temp.Observe(rValue);
    _temp.WithSpan(_spn);    // pin _spn on the next flush
    _spn.End();              // span closes, but frame still carries its ID
*)
METHOD PUBLIC WithSpan : BOOL
VAR_INPUT
    pSpan : REFERENCE TO FB_Span;
END_VAR
_pSpanOverride REF= pSpan;
WithSpan := TRUE;
END_METHOD

END_FUNCTION_BLOCK

// ---- POUs/Metrics/FB_TcOtelTaskMetrics.TcPOU
(*
:Description: Per-task transport for FB_Metrics push frames — queued, zero-copy.

INTERNAL — never instantiated by user code. One instance per task lives in
``PRG_TaskLog.aTaskMetrics`` and is driven once per cycle by
``PRG_TaskLog.Call()``. Owns the ``ADSWRITE`` FB that ships pre-assembled
metric frames to ``IG = 0x4D424301`` / ``IO = 2`` (IO_PUSH_METRIC_AGG).

**Phase 8: queued dispatch instead of single-flight drop.**

Multiple FB_Metrics instances on the same task routinely flush in the same
window (e.g. two metrics both at 5 s push interval). The previous version
single-flighted ADSWRITE and dropped every concurrent Emit — the second
metric lost its frame. This version keeps a small ring of POINTER TO
FB_Metrics and drives ADSWRITE through them one at a time.

The sender never copies the frame. FB_Metrics lays out its header + body in
a single contiguous buffer (header grows backward into a 256-byte reserve
right before the body). On enqueue the sender grabs ``_GetPendingPtr`` +
``_GetPendingLen`` from the FB; ADSWRITE reads directly from the FB's own
memory. On completion the sender calls ``_NotifyFrameSent`` so the FB
releases its pending half and either resumes collecting into it or drops
the next window if the sender has fallen behind.

Watchdog mirrors ``FB_TcOtelTaskDiag`` — if ADSWRITE.BUSY stays true past
``nFlightWatchdogCycles`` the in-flight frame is cut loose (``WRITE := FALSE``)
so a transient tc-otel outage doesn't wedge the sender forever.

Ring overflow (``nCount = SIZEOF_RING``) is the only remaining drop path.
It means ADSWRITE is grinding through a backlog deeper than the ring. In
normal operation ``nFlushDropCount`` should stay at 0; a non-zero value
signals either a dead tc-otel endpoint or a massive burst of FBs flushing
simultaneously on one task.
*)
{attribute 'no_explicit_call' := 'no direct call necessary'}
{attribute 'conditionalshow'}
FUNCTION_BLOCK INTERNAL FB_TcOtelTaskMetrics
VAR CONSTANT
    (* Queue depth. 8 covers up to 8 FB_Metrics flushing on the same cycle
       before any drop. Memory cost = 8 * SIZEOF(POINTER) ≈ 32-64 B. *)
    SIZEOF_RING             : UDINT := 8;
END_VAR
VAR
    bInitialized            : BOOL;
    sTcOtelNetId            : T_AmsNetId;
    nTcOtelPort             : UINT := 16150;

    (* Wire constants — matches diagnostics.rs IG_PUSH_DIAG / IO_PUSH_METRIC_AGG. *)
    nIdxGroupPushDiag       : UDINT := 16#4D424301;
    nIdxOffsetMetricAgg     : UDINT := 2;

    (* ADS write state. Zero-copy: SRCADDR points directly into whichever
       FB_Metrics frame half is pending. *)
    fbAdsWrite              : Tc2_System.ADSWRITE;
    bFlushInFlight          : BOOL;
    (* Identity-critical: compared against ring slots (POINTER TO FB_Metrics)
       during Dequeue. Kept as POINTER because ADR() of a REFERENCE returns
       the reference-storage address, not the target — which would never
       match the target address stored in the ring. *)
    pInFlight               : POINTER TO FB_Metrics;
    nFlushStartCycle        : UDINT;
    nFlightWatchdogCycles   : UDINT := 2000;
    nLastFlushSuccessCycle  : UDINT;

    (* Per-task enqueue ring — FIFO of FB_Metrics waiting to ship. *)
    aPending                : ARRAY[0..7] OF POINTER TO FB_Metrics;
    nPendingHead            : UDINT;
    nPendingTail            : UDINT;
    nPendingCount           : UDINT;

    (* Ops counters. *)
    nFlushDropCount         : UDINT;     // ring overflow — real drops
    nFlushErrorCount        : UDINT;     // ADSWRITE returned ERR
    nFlushOkCount           : UDINT;     // successful ships
    nPendingHighWater       : UDINT;     // peak nPendingCount since boot
END_VAR

(*
:Description: Start ADSWRITE for the head of the pending ring.

No-op when a flush is already in flight or when the ring is empty. Reads
the pending frame's byte pointer and length directly from the FB_Metrics
instance (zero-copy) and arms the ADSWRITE FB with rising-edge WRITE.
*)
METHOD PRIVATE _KickHead
VAR
    pHead     : POINTER TO FB_Metrics;
    pFb       : REFERENCE TO FB_Metrics;
    pSrc      : PVOID;
    nLen      : UDINT;
    nTaskIdx  : DINT;
    nNowCycle : UDINT;
END_VAR
IF bFlushInFlight OR nPendingCount = 0 OR NOT bInitialized THEN
    RETURN;
END_IF

(* Peek-then-pop: read the head slot FIRST, then clear it and advance.
   Reordering these three writes corrupts the queue — the defensive check
   below only fires when the enqueue itself was buggy. *)
pHead := aPending[nPendingHead];
aPending[nPendingHead] := 0;
nPendingHead  := (nPendingHead + 1) MOD SIZEOF_RING;
nPendingCount := nPendingCount - 1;

IF pHead = 0 THEN
    (* Defensive — should not happen with well-formed enqueue/dequeue. *)
    RETURN;
END_IF
pFb REF= pHead^;

(* Ask the FB for the pending frame's byte pointer + length. *)
pSrc := pFb._GetPendingPtr();
nLen := pFb._GetPendingLen();
IF pSrc = 0 OR nLen = 0 THEN
    (* FB had nothing pending — the enqueue was spurious. Notify with
       success so the FB resets its pending state, then try the next. *)
    pFb._NotifyFrameSent(TRUE);
    _KickHead();
    RETURN;
END_IF

(* Rising-edge ADSWRITE kick — same idiom as FB_TcOtelTask. *)
fbAdsWrite(WRITE := FALSE);
fbAdsWrite(
    NETID   := sTcOtelNetId,
    PORT    := nTcOtelPort,
    IDXGRP  := nIdxGroupPushDiag,
    IDXOFFS := nIdxOffsetMetricAgg,
    LEN     := nLen,
    SRCADDR := pSrc,
    WRITE   := TRUE,
    TMOUT   := T#1S
);

pInFlight        := pHead;
bFlushInFlight   := TRUE;

nTaskIdx  := Tc2_Utilities.GETCURTASKINDEXEX();
IF nTaskIdx > 0 THEN
    nNowCycle        := TwinCAT_SystemInfoVarList._TaskInfo[nTaskIdx].CycleCount;
    nFlushStartCycle := nNowCycle;
END_IF
END_METHOD

(*
:Description: Pump in-flight ADSWRITE — drives flush completion + watchdog.

Called once per task cycle from ``PRG_TaskLog.Call()``. Cheap when the
queue is empty. On ADSWRITE completion the FB that owned the frame is
notified (so it can release its pending half) and the next queued frame
is kicked off immediately within the same cycle — no cycle-delay between
back-to-back frames.
*)
METHOD PUBLIC Call
VAR
    nTaskIdx   : DINT;
    nNowCycle  : UDINT;
    pCompleted : POINTER TO FB_Metrics;
    bOk        : BOOL;
END_VAR
IF NOT bFlushInFlight THEN
    RETURN;
END_IF

fbAdsWrite();

nTaskIdx  := Tc2_Utilities.GETCURTASKINDEXEX();
nNowCycle := TwinCAT_SystemInfoVarList._TaskInfo[nTaskIdx].CycleCount;

IF NOT fbAdsWrite.BUSY THEN
    bOk := NOT fbAdsWrite.ERR;
    IF bOk THEN
        nFlushOkCount          := nFlushOkCount + 1;
        nLastFlushSuccessCycle := nNowCycle;
    ELSE
        nFlushErrorCount := nFlushErrorCount + 1;
    END_IF

    (* Notify the FB first (so it can release its pending half), THEN
       clear our in-flight latch, THEN kick the next queued frame. *)
    pCompleted     := pInFlight;
    pInFlight      := 0;
    bFlushInFlight := FALSE;
    fbAdsWrite(WRITE := FALSE);

    IF pCompleted <> 0 THEN
        pCompleted^._NotifyFrameSent(bOk);
    END_IF

    _KickHead();

ELSIF nFlushStartCycle <> 0
    AND (nNowCycle - nFlushStartCycle) > nFlightWatchdogCycles THEN
    (* Watchdog tripped — cut the wedged call loose so later pushes can
       still reach tc-otel when connectivity is restored. Notify the FB
       with failure so its pending half is freed anyway. *)
    nFlushErrorCount := nFlushErrorCount + 1;
    pCompleted     := pInFlight;
    pInFlight      := 0;
    bFlushInFlight := FALSE;
    fbAdsWrite(WRITE := FALSE);

    IF pCompleted <> 0 THEN
        pCompleted^._NotifyFrameSent(FALSE);
    END_IF

    _KickHead();
END_IF
END_METHOD

(*
:Description: Remove every pending entry for ``pFb`` from the ring.

Called from ``FB_Metrics.FB_exit`` so a destroyed instance can't leave a
stale pointer in the ring. Safe to call when the FB is in-flight — in that
case the pending ring is already clean but ``pInFlight`` is cleared and
ADSWRITE is cut loose to prevent a post-destruction SRCADDR read. Linear
scan; ring depth is small.
*)
METHOD PUBLIC Dequeue
VAR_INPUT
    pFb : POINTER TO FB_Metrics;
END_VAR
VAR
    nRead   : UDINT;
    nWrite  : UDINT;
    nKept   : UDINT;
    i       : UDINT;
END_VAR
IF pFb = 0 THEN
    RETURN;
END_IF

(* Compact in place: iterate head→tail, drop entries whose pointer equals pFb.
   Identity by raw address — ring slots and pInFlight both store target-of-FB
   addresses. Using REFERENCE TO with ADR() wouldn't work here because ADR
   on a REFERENCE returns the reference-storage address, not the target's. *)
nKept := 0;
FOR i := 0 TO nPendingCount - 1 DO
    nRead := (nPendingHead + i) MOD SIZEOF_RING;
    IF aPending[nRead] <> pFb THEN
        IF nKept <> i THEN
            nWrite := (nPendingHead + nKept) MOD SIZEOF_RING;
            aPending[nWrite] := aPending[nRead];
        END_IF
        nKept := nKept + 1;
    END_IF
END_FOR

(* Zero out the tail slots left behind. *)
FOR i := nKept TO nPendingCount - 1 DO
    nWrite := (nPendingHead + i) MOD SIZEOF_RING;
    aPending[nWrite] := 0;
END_FOR

nPendingCount := nKept;
nPendingTail  := (nPendingHead + nKept) MOD SIZEOF_RING;

(* If the destroyed FB is currently being shipped, cut ADSWRITE loose
   without notifying — the FB is gone, notification would double-free.
   nFlushOkCount / nFlushErrorCount stay unchanged since the outcome is
   unknown and the frame is being abandoned mid-flight. *)
IF bFlushInFlight AND pInFlight = pFb THEN
    fbAdsWrite(WRITE := FALSE);
    pInFlight      := 0;
    bFlushInFlight := FALSE;
END_IF
END_METHOD

(*
:Description: Queue ``pFb`` for next ADSWRITE dispatch.

Returns FALSE only when the ring is already full (real overflow — should
stay near zero; signals sender backlog). Returns TRUE on successful enqueue
and, if the sender is idle, kicks the head immediately so single-enqueue
scenarios ship within the same cycle.

The caller (``FB_Metrics._DoFlush``) must guarantee that the pending half
stays stable until ``_NotifyFrameSent`` is called back.
*)
METHOD PUBLIC Enqueue : BOOL
VAR_INPUT
    pFb : POINTER TO FB_Metrics;
END_VAR
IF NOT bInitialized OR pFb = 0 THEN
    Enqueue := FALSE;
    RETURN;
END_IF

IF nPendingCount >= SIZEOF_RING THEN
    nFlushDropCount := nFlushDropCount + 1;
    Enqueue := FALSE;
    RETURN;
END_IF

aPending[nPendingTail] := pFb;
nPendingTail  := (nPendingTail + 1) MOD SIZEOF_RING;
nPendingCount := nPendingCount + 1;

IF nPendingCount > nPendingHighWater THEN
    nPendingHighWater := nPendingCount;
END_IF

(* If sender is idle, fire immediately so small loads ship without a
   cycle delay. If busy, Call() will kick the head on completion. *)
IF NOT bFlushInFlight THEN
    _KickHead();
END_IF

Enqueue := TRUE;
END_METHOD

(*
:Description: Bind this sender to a tc-otel endpoint.

Safe to call repeatedly — overwrites the previous endpoint. Call from
``PRG_TaskLog.Init`` so every task that runs ``PRG_TaskLog.Call()`` has
its metric sender initialized.
*)
METHOD PUBLIC Init : BOOL
VAR_INPUT
    sAmsNetId : T_AmsNetId;
    nPort     : UINT;     // tc-otel ADS port; 0 keeps the default 16150
END_VAR
sTcOtelNetId := sAmsNetId;
IF nPort <> 0 THEN
    nTcOtelPort := nPort;
END_IF
bInitialized := TRUE;
Init := TRUE;
END_METHOD

(*
:Description: TRUE while ADSWRITE is shipping a frame.

Surfaced for diagnostics / tests. Not consulted by FB_Metrics (Enqueue
always succeeds unless the ring is full).
*)
PROPERTY PUBLIC IsBusy : BOOL
GET
IsBusy := bFlushInFlight;
END_GET
END_PROPERTY

(*
:Description: Current number of pending frames in the dispatch ring
(not counting the in-flight frame, if any).
*)
PROPERTY PUBLIC QueueDepth : UDINT
GET
QueueDepth := nPendingCount;
END_GET
END_PROPERTY

END_FUNCTION_BLOCK

// ---- API/Trace/F_TraceParentFromString.TcPOU
(*
:Description: Build a W3C traceparent header by hashing domain identifiers
into the trace_id and (optional) parent_span_id positions.

Returns the canonical 55-char string ``00-<trace>-<span>-01`` where:

* ``<trace>`` is ``F_HashTraceId(sTraceId)`` — a 32-hex digest of any
  domain identifier naming the trace (workpiece ID, order ID, session
  ID, …). Every PLC that hashes the same ``sTraceId`` produces the
  same trace_id, so their spans aggregate under one trace in Tempo
  without any explicit traceparent handoff.
* ``<span>`` is ``F_HashSpanId(sParentId)`` when ``sParentId`` is
  non-empty, or 16 zeros when empty. The all-zero form is the
  OTel-defined "no parent" marker; tc-otel treats the consumer span
  as root within its trace.

Typical use: **brownfield aggregation** where MES / DB / barcode gives
you a business identifier (order_id, workpiece_id, batch_id) but not
a pre-minted traceparent. Every station hashing the same sTraceId
aggregates its spans into one Tempo trace.

Example (aggregation-only; sibling spans under one trace_id):

    sTp := F_TraceParentFromString(sTraceId := 'WP-1234');
    spn.Begin(sName := 'station_weigh', sTraceParent := sTp);

Example (explicit chain — consumer cites an upstream producer):

    sTp := F_TraceParentFromString(
        sTraceId  := 'WP-1234',
        sParentId := 'station_weigh');          // name of upstream span
    spn.Begin(sName := 'station_inspect', sTraceParent := sTp);

For true distributed tracing with a transport carrying traceparent
between producers and consumers, prefer forwarding
``PRG_TaskLog.Span.CurrentTraceParent()`` — it returns the exact bytes
tc-otel stored, so multi-hop chains stay consistent without relying
on hash agreement.
*)
FUNCTION F_TraceParentFromString : STRING(60)
VAR_INPUT
    sTraceId  : STRING(80);                 (* identifier hashed via F_HashTraceId → 32-hex trace_id *)
    sParentId : STRING(80) := '';           (* identifier hashed via F_HashSpanId → 16-hex span_id;
                                               empty = no parent (all-zero span_id) *)
END_VAR
VAR
    sTraceHex : STRING(32);
    sSpanHex  : STRING(16);
END_VAR


sTraceHex := F_HashTraceId(sTraceId);

(* Validate sender span_id: must be exactly 16 hex chars, otherwise
   fall back to the all-zero "no parent" marker. This keeps malformed
   callers from producing invalid W3C headers that tc-otel would
   reject. *)
   
IF sParentId <> '' THEN
    sSpanHex := F_HashSpanId(sParentId);
ELSE
    sSpanHex := '0000000000000000';  (* W3C: all-zero span_id = "invalid", signals no parent *)
END_IF

F_TraceParentFromString := CONCAT(
    CONCAT(
        CONCAT('00-', sTraceHex),
        CONCAT('-', sSpanHex)),
    '-01');

END_FUNCTION

// ---- POUs/Trace/F_HashTraceId.TcPOU
(*
:Description: Deterministic 128-bit hash of an arbitrary domain
identifier, rendered as 32 lowercase hex characters for use as a W3C
trace_id.

Every PLC that hashes the same ``sTraceId`` input (workpiece ID,
order ID, session ID, …) produces the same hex string, enabling
trace aggregation across modules that share only the domain
identifier and no explicit traceparent handoff (Pattern D in
docs/traces-propagation.md — transport-less cross-PLC tracing via
barcode / RFID / conveyor routing).

Internal — callers should use ``F_TraceParentFromString`` to build a
complete traceparent header. Direct use of this hash is only
appropriate when the caller already has the W3C framing.

Implementation: two parallel xorshift64 streams seeded from different
constants, folded over the input bytes. Collision probability for
distinct 80-char inputs is ~1/2^128 — adequate for OTel trace_id use
(spec requires "randomly generated", not cryptographic). Deterministic
across PLC reboots and runtime reloads.
*)
FUNCTION INTERNAL F_HashTraceId : STRING(32)
VAR_INPUT
    sTraceId : STRING(80);   (* any domain identifier — workpiece, order, session, ... *)
END_VAR
VAR
    i         : INT;
    nLen      : INT;
    hi        : ULINT;
    lo        : ULINT;
    b         : BYTE;
    nNibble   : BYTE;
    achHex    : ARRAY[0..15] OF BYTE := [16#30, 16#31, 16#32, 16#33, 16#34, 16#35, 16#36, 16#37, 16#38, 16#39, 16#61, 16#62, 16#63, 16#64, 16#65, 16#66];
    achOut    : ARRAY[0..31] OF BYTE;
    achResult : STRING(32);
END_VAR


(* Two independent seeds so the upper and lower 64 bits of the 128-bit
   digest can't collapse to the same value for any input. *)
hi := 16#9E3779B97F4A7C15;
lo := 16#C6BC279692B5C323;

nLen := TO_INT(Tc2_Utilities.LEN2(ADR(sTraceId)));
IF nLen > 80 THEN
    nLen := 80;
END_IF;

(* Fold each byte into both streams, then advance xorshift64 once per
   byte so position matters (order-sensitive hash). *)
FOR i := 0 TO nLen - 1 DO
    b := sTraceId[i];
    hi := hi XOR TO_ULINT(b);
    hi := hi XOR SHL(hi, 13);
    hi := hi XOR SHR(hi, 7);
    hi := hi XOR SHL(hi, 17);

    lo := lo XOR (TO_ULINT(b) * 16#100000001B3);
    lo := lo XOR SHL(lo, 11);
    lo := lo XOR SHR(lo, 5);
    lo := lo XOR SHL(lo, 23);
END_FOR

(* Write digest LE: hi → bytes 0..7, lo → bytes 8..15. Then hex-encode. *)
FOR i := 0 TO 7 DO
    achOut[i]     := 0;  (* placeholder, filled below *)
END_FOR
Tc2_System.MEMCPY(ADR(achOut[0]), ADR(hi), 8);
Tc2_System.MEMCPY(ADR(achOut[8]), ADR(lo), 8);

(* Emit 32 hex chars into a STRING(32). Two chars per byte, 16 bytes total. *)
FOR i := 0 TO 15 DO
    b := achOut[i];
    nNibble := SHR(b, 4) AND 16#0F;
    achResult[i * 2]     := achHex[nNibble];
    nNibble := b AND 16#0F;
    achResult[i * 2 + 1] := achHex[nNibble];
END_FOR
achResult[32] := 0;

F_HashTraceId := achResult;

END_FUNCTION

// ---- POUs/Trace/F_HashSpanId.TcPOU
(*
:Description: Deterministic 64-bit hash of a sender/span identifier,
rendered as 16 lowercase hex characters for use as a W3C parent_id
(span-id) in a traceparent header. Every PLC that calls this function
with the same ``sSpanId`` produces the same hex string, so the sender's
emitted span_id and the receiver's parent_id match up without an
explicit traceparent handoff (Pattern D — transport-less cross-PLC
tracing via barcode / RFID / conveyor routing).
Implementation: single xorshift64 stream, seeded from a constant that
differs from ``F_HashTraceId`` so that trace_id and span_id derived
from the same input don't share byte patterns. Collision probability
for distinct inputs is ~1/2^64 — adequate for OTel span_id use (spec
requires "randomly generated", not cryptographic). Deterministic
across PLC reboots and runtime reloads.
*)
FUNCTION INTERNAL F_HashSpanId : STRING(16)
VAR_INPUT
    sSpanId : STRING(80);
END_VAR
VAR
    i         : INT;
    nLen      : INT;
    h         : ULINT;
    b         : BYTE;
    nNibble   : BYTE;
    achHex    : ARRAY[0..15] OF BYTE := [16#30, 16#31, 16#32, 16#33, 16#34, 16#35, 16#36, 16#37, 16#38, 16#39, 16#61, 16#62, 16#63, 16#64, 16#65, 16#66];
    achOut    : ARRAY[0..7] OF BYTE;
    achResult : STRING(16);
END_VAR

(* Seed deliberately different from F_HashTraceId's hi/lo constants so
   span_id and trace_id hashed from the same input can't collide on
   bytes. *)
h := 16#D1B54A32D192ED03;
nLen := TO_INT(Tc2_Utilities.LEN2(ADR(sSpanId)));
IF nLen > 80 THEN
    nLen := 80;
END_IF;
(* Fold each byte into the stream, then advance xorshift64 once per
   byte so position matters (order-sensitive hash). *)
FOR i := 0 TO nLen - 1 DO
    b := sSpanId[i];
    h := h XOR TO_ULINT(b);
    h := h XOR SHL(h, 13);
    h := h XOR SHR(h, 7);
    h := h XOR SHL(h, 17);
END_FOR
Tc2_System.MEMCPY(ADR(achOut[0]), ADR(h), 8);
(* Emit 16 hex chars into a STRING(16). Two chars per byte, 8 bytes total. *)
FOR i := 0 TO 7 DO
    b := achOut[i];
    nNibble := SHR(b, 4) AND 16#0F;
    achResult[i * 2]     := achHex[nNibble];
    nNibble := b AND 16#0F;
    achResult[i * 2 + 1] := achHex[nNibble];
END_FOR
achResult[16] := 0;
F_HashSpanId := achResult;

END_FUNCTION

// ---- POUs/Diagnostic/FB_TcOtelTaskDiag.TcPOU
(*
:Description: Per-task push-diagnostic collector.

One instance per task lives in ``PRG_TaskLog.aTaskDiag`` and is driven
once per cycle by ``PRG_TaskLog.Call()``. Each cycle the FB captures a
``ST_PushDiagSample`` (cycle_count, exec_time, dc_time, flags) into a
1024-entry ring buffer. When the aggregation window expires it flushes
the ring plus the window's aggregates (min/max/avg exec time,
exceed/rtv counts) as a single batch frame via ``ADSWRITE`` to tc-otel.

Operators tune the window through ``PRG_TaskLog.aTaskDiagConfig`` which
tc-otel writes via ADS symbol access.
*)
{attribute 'no_explicit_call' := 'no direct call necessary'}
{attribute 'conditionalshow'}
FUNCTION_BLOCK INTERNAL FB_TcOtelTaskDiag
VAR_INPUT
END_VAR
VAR
    bInitialized        : BOOL;
    sTcOtelNetId        : T_AmsNetId;
    nTcOtelPort         : UINT := 16150;
    pConfig             : REFERENCE TO ST_PushDiagConfig;

    (* Wire-format constants — kept as VAR to avoid a separate GVL. *)
    nWireVersion        : BYTE  := 2;
    nEventTypeBatch     : BYTE  := 10;
    nHeaderSize         : UDINT  := 80;
    nSampleSize         : UDINT  := 24;
    nMaxSamples         : UDINT  := 1024;
    nFlagCycleExceed    : BYTE  := 1;
    nFlagRtViolation    : BYTE  := 2;
    nFlagFirstCycle     : BYTE  := 4;
    nFlagOverflow       : BYTE  := 8;
    nIdxGroupPushDiag   : UDINT := 16#4D424301;
    nIdxOffsetBatch     : UDINT := 0;

    (* Ring buffer — 1024 samples, ~24 KB per task instance. *)
    aSampleRing         : ARRAY [0..1023] OF ST_PushDiagSample;
    nRingHead           : UDINT;     // next write slot
    nRingCount          : UDINT;     // samples currently in the ring
    bOverflowPending    : BOOL;      // next stored sample carries the overflow flag

    (* Per-window aggregates. Cleared after each flush. *)
    nExecTimeMinUs      : UDINT;
    nExecTimeMaxUs      : UDINT;
    nExecTimeSumUs      : ULINT;
    nExecTimeSamples    : UDINT;
    nCycleExceedInWnd   : UDINT;
    nRtViolationInWnd   : UDINT;
    nCycleCountStart    : UDINT;
    nCycleCountEnd      : UDINT;
    nDcTimeStart        : LINT;
    nDcTimeEnd          : LINT;
    bWindowHasSample    : BOOL;
    nWindowStartCycle   : UDINT;
    bWindowStartSet     : BOOL;

    (* Divider state for sub-sampling. *)
    nDividerCounter     : USINT;

    (* RTViolation is an edge-like event — keep rising-edge detection to
       avoid double-counting. CycleTimeExceeded is a per-cycle condition
       (task exec > cycle time for THAT cycle) so we count every TRUE
       cycle, matching what XAE's Exceed Counter shows. *)
    bPrevRtViolation      : BOOL;

    (* Lifetime exceed counters — never reset per window. Visible in the
       online view so you can compare directly against XAE's per-task
       Exceed column and confirm the detection logic actually fires. *)
    nLifetimeExceedCount  : UDINT;
    nLifetimeRtvCount     : UDINT;
    nMaxExecTimeUs        : UDINT;
    nLastExecTimeUs       : UDINT;
    nLastCycleTimeUs      : UDINT;

    (* ADS write state. The watchdog guards against a permanently-stuck
       ADSWRITE (e.g. tc-otel unreachable) — after nFlightWatchdogCycles
       have elapsed since the flush was kicked, the FB force-resets
       WRITE:=FALSE and drops the batch. Cycle-count based like the
       window timer so the two agree on "elapsed time". *)
    fbAdsWrite              : Tc2_System.ADSWRITE;
    bFlushInFlight          : BOOL;
    nFlushStartCycle        : UDINT;
    nFlightWatchdogCycles   : UDINT := 2000;
    nLastFlushSuccessCycle  : UDINT;
    nFlushDropCount         : UDINT;
    nFlushErrorCount        : UDINT;
    nFlushOkCount           : UDINT;

    (* Scratch for (de)serialization. *)
    stHeader            : ST_PushDiagBatchHeader;
    abySendBuffer       : ARRAY [0..24655] OF BYTE;  // 80 + 1024 * 24
END_VAR

(*
:Description: Capture one cycle's diagnostic sample and flush on window expiry.

Called once per task cycle from ``PRG_TaskLog.Call()``. Cheap — ~20 lines
of straight-line code on the sample path. Flush only fires when the
configured window has elapsed.
*)
METHOD PUBLIC Call
VAR_INPUT
END_VAR
VAR
    nTaskIdx            : DINT;
    pTaskInfo           : POINTER TO PlcTaskSystemInfo;
    stSample            : ST_PushDiagSample;
    nFlags              : BYTE;
    nExecNow            : UDINT;
    nRequestedDivider   : USINT;
END_VAR
(* This FB lives as an array element in PRG_TaskLog and is never invoked
   directly — only Call() runs each cycle. Every state transition that
   normally belongs in the FB body (ADSWRITE pumping especially) has to
   happen here. Same pattern the logger's FB_TcOtelTask uses.

   Watchdog: if ADSWRITE's BUSY stays true past nFlightWatchdogCycles the
   current batch is abandoned (WRITE:=FALSE resets the FB), bFlushInFlight
   is cleared, and the next window is allowed to flush normally. Without
   this guard a transient tc-otel outage wedges the FB forever because
   nothing else clears bFlushInFlight. *)
IF bFlushInFlight THEN
    fbAdsWrite();
    IF NOT fbAdsWrite.BUSY THEN
        IF fbAdsWrite.ERR THEN
            nFlushErrorCount := nFlushErrorCount + 1;
        ELSE
            nFlushOkCount          := nFlushOkCount + 1;
            nLastFlushSuccessCycle := TwinCAT_SystemInfoVarList._TaskInfo[
                                         Tc2_Utilities.GETCURTASKINDEXEX()].CycleCount;
        END_IF
        fbAdsWrite(WRITE := FALSE);
        bFlushInFlight := FALSE;
    ELSIF nFlushStartCycle <> 0
        AND (TwinCAT_SystemInfoVarList._TaskInfo[
                 Tc2_Utilities.GETCURTASKINDEXEX()].CycleCount - nFlushStartCycle)
             > nFlightWatchdogCycles THEN
        (* Watchdog tripped — cut the wedged call loose so later windows
           can still reach tc-otel when connectivity is restored. *)
        nFlushDropCount := nFlushDropCount + 1;
        fbAdsWrite(WRITE := FALSE);
        bFlushInFlight := FALSE;
    END_IF
END_IF

IF NOT bInitialized OR NOT __ISVALIDREF(pConfig) THEN
    RETURN;
END_IF

IF NOT pConfig.enabled THEN
    RETURN;
END_IF

(* Divider: skip cycles if configured to sub-sample a very fast task. *)
nRequestedDivider := pConfig.divider;
IF nRequestedDivider > 1 THEN
    nDividerCounter := nDividerCounter + 1;
    IF nDividerCounter < nRequestedDivider THEN
        (* still check window expiry even on skipped cycles *)
        THIS^.CheckFlush();
        RETURN;
    END_IF
    nDividerCounter := 0;
END_IF

(* Resolve our task info. *)
nTaskIdx := Tc2_Utilities.GETCURTASKINDEXEX();
IF nTaskIdx <= 0 THEN
    RETURN;
END_IF
pTaskInfo := ADR(TwinCAT_SystemInfoVarList._TaskInfo[nTaskIdx]);

(* Build the sample.
   dc_time uses `DcTaskTime` — the DC clock stamped at the start of THIS
   task cycle (LINT, nanoseconds). That gives cycle-granular timestamps
   (not the ~100 ms-quantised RtcTime), so every sample lands at its true
   cycle time on the Grafana axis and matches log correlation to the
   nanosecond. DcTaskTime is already an int64 ns-since-epoch (DC-synced),
   so no FILETIME conversion needed — but the wire field layout is the
   same LINT, and tc-otel's filetime_to_datetime handles either by
   treating the value as 100 ns ticks since 1601 for FILETIME-style and
   directly for DC-style when the value is below the FILETIME epoch
   offset. To keep the wire format unambiguous we ship DcTaskTime raw
   and let the Rust side decide. *)
stSample.cycle_count  := pTaskInfo^.CycleCount;
nExecNow              := pTaskInfo^.LastExecTime;
stSample.exec_time_us := nExecNow;
stSample.dc_time      := pTaskInfo^.DcTaskTime;

nFlags := 0;

(* Expose a few raw TaskInfo values on the instance so the online view
   matches exactly what we sample. Values in microseconds (TaskInfo
   fields are 100 ns ticks). *)
nLastCycleTimeUs := pTaskInfo^.CycleTime / 10;
nLastExecTimeUs  := nExecNow / 10;
IF nLastExecTimeUs > nMaxExecTimeUs THEN
    nMaxExecTimeUs := nLastExecTimeUs;
END_IF

(* CycleTimeExceeded: count every cycle where the flag is TRUE. The
   runtime sets it once per cycle that exceeded, so a 5-cycle exceed
   burst contributes 5 counts — matches XAE's per-cycle semantics. *)
IF pTaskInfo^.CycleTimeExceeded THEN
    nCycleExceedInWnd    := nCycleExceedInWnd + 1;
    nLifetimeExceedCount := nLifetimeExceedCount + 1;
    nFlags               := nFlags OR nFlagCycleExceed;
END_IF

(* RT violation stays edge-triggered — it represents a discrete event
   rather than a condition, and the runtime may latch it for a short
   window after the fact. *)
IF pTaskInfo^.RTViolation AND NOT bPrevRtViolation THEN
    nRtViolationInWnd := nRtViolationInWnd + 1;
    nLifetimeRtvCount := nLifetimeRtvCount + 1;
    nFlags            := nFlags OR nFlagRtViolation;
END_IF
bPrevRtViolation := pTaskInfo^.RTViolation;
IF pTaskInfo^.FirstCycle THEN
    nFlags := nFlags OR nFlagFirstCycle;
END_IF
IF bOverflowPending THEN
    nFlags := nFlags OR nFlagOverflow;
    bOverflowPending := FALSE;
END_IF
stSample.flags := nFlags;

(* Store the sample. Ring wraps; on overflow we mark the NEXT sample so
   tc-otel sees the gap without having to infer it from cycle_count. *)
aSampleRing[nRingHead] := stSample;
nRingHead := nRingHead + 1;
IF nRingHead >= nMaxSamples THEN
    nRingHead := 0;
END_IF
IF nRingCount < nMaxSamples THEN
    nRingCount := nRingCount + 1;
ELSE
    (* Ring was already full — oldest sample just got overwritten. *)
    bOverflowPending := TRUE;
END_IF

(* Update aggregates. *)
IF NOT bWindowHasSample THEN
    nExecTimeMinUs    := nExecNow;
    nExecTimeMaxUs    := nExecNow;
    nCycleCountStart  := stSample.cycle_count;
    nDcTimeStart      := stSample.dc_time;
    bWindowHasSample  := TRUE;
ELSE
    IF nExecNow < nExecTimeMinUs THEN
        nExecTimeMinUs := nExecNow;
    END_IF
    IF nExecNow > nExecTimeMaxUs THEN
        nExecTimeMaxUs := nExecNow;
    END_IF
END_IF
nCycleCountEnd   := stSample.cycle_count;
nDcTimeEnd       := stSample.dc_time;
nExecTimeSumUs   := nExecTimeSumUs + UDINT_TO_ULINT(nExecNow);
nExecTimeSamples := nExecTimeSamples + 1;

THIS^.CheckFlush();
END_METHOD

(*
:Description: Internal — flush the ring if the aggregation window elapsed.

Kept on the happy-path so timer checks don't inflate Call() itself.
*)
METHOD PRIVATE CheckFlush
VAR_INPUT
END_VAR
VAR
    nNowCycle      : UDINT;
    nDeltaCycles   : UDINT;
    nTargetCycles  : UDINT;
    nCycleTimeUs   : UDINT;
    pTi            : POINTER TO PlcTaskSystemInfo;
    nTi            : DINT;
END_VAR
IF NOT __ISVALIDREF(pConfig) OR pConfig.window_ms = 0 THEN
    RETURN;
END_IF

(* Window timing is cycle-count based — CycleCount is a pure monotonic
   task counter incremented once per cycle by the TwinCAT runtime. That
   is the most reliable "time" source we have inside a PLC task:
     - no jitter (unlike RtcTime / FILETIME which reset on sync)
     - no drift (unlike accumulating delta times)
     - cycle-exact alignment with the batched samples
   A 100 ms window at 1 ms task cycle flushes every 100 cycles, period. *)
nTi := Tc2_Utilities.GETCURTASKINDEXEX();
IF nTi <= 0 THEN
    RETURN;
END_IF
pTi := ADR(TwinCAT_SystemInfoVarList._TaskInfo[nTi]);

(* CycleTime in PlcTaskSystemInfo is in 100 ns units; convert to µs
   so target_cycles = window_ms * 1000 / cycle_time_us is clean. *)
nCycleTimeUs := pTi^.CycleTime / 10;
IF nCycleTimeUs = 0 THEN
    nCycleTimeUs := 1000; (* safety fallback: assume 1 ms *)
END_IF
nTargetCycles := (pConfig.window_ms * 1000) / nCycleTimeUs;
IF nTargetCycles = 0 THEN
    nTargetCycles := 1;
END_IF

nNowCycle := pTi^.CycleCount;
IF NOT bWindowStartSet OR nNowCycle < nWindowStartCycle THEN
    nWindowStartCycle := nNowCycle;
    bWindowStartSet   := TRUE;
    RETURN;
END_IF
nDeltaCycles := nNowCycle - nWindowStartCycle;
IF nDeltaCycles < nTargetCycles THEN
    RETURN;
END_IF

IF NOT bWindowHasSample OR bFlushInFlight THEN
    nWindowStartCycle := nNowCycle;
    RETURN;
END_IF

THIS^.Flush();
nWindowStartCycle := nNowCycle;
END_METHOD

(*
:Description: Internal — serialize the ring + aggregates and kick ADSWRITE.

No-op when the ring is empty or a previous write is still in flight.
*)
METHOD PRIVATE Flush
VAR_INPUT
END_VAR
VAR
    nStartRead    : UDINT;
    nOffset       : UDINT;
    nLocalIdx     : UDINT;
    nRingIter     : UDINT;
    pTask         : POINTER TO PlcTaskSystemInfo;
    nTi           : DINT;
    nNameLen      : UDINT;
    sTaskName     : STRING;
    nBytesToWrite : UDINT;
END_VAR
IF bFlushInFlight OR nRingCount = 0 THEN
    RETURN;
END_IF

(* Resolve task info for task_obj_id / port / name. *)
nTi := Tc2_Utilities.GETCURTASKINDEXEX();
IF nTi <= 0 THEN
    RETURN;
END_IF
pTask := ADR(TwinCAT_SystemInfoVarList._TaskInfo[nTi]);

(* Build header. *)
stHeader.version            := nWireVersion;
stHeader.event_type         := nEventTypeBatch;
stHeader.reserved0          := 0;
stHeader.task_obj_id        := pTask^.ObjId;
stHeader.task_port          := DWORD_TO_UINT(pTask^.AdsPort AND 16#FFFF);
stHeader.window_ms          := UDINT_TO_UINT(pConfig.window_ms);
stHeader.sample_count       := UDINT_TO_UINT(nRingCount);
stHeader.reserved1          := 0;
stHeader.cycle_count_start  := nCycleCountStart;
stHeader.cycle_count_end    := nCycleCountEnd;
stHeader.dc_time_start      := nDcTimeStart;
stHeader.dc_time_end        := nDcTimeEnd;
stHeader.exec_time_min_us   := nExecTimeMinUs;
stHeader.exec_time_max_us   := nExecTimeMaxUs;
IF nExecTimeSamples > 0 THEN
    stHeader.exec_time_avg_us := ULINT_TO_UDINT(nExecTimeSumUs / UDINT_TO_ULINT(nExecTimeSamples));
ELSE
    stHeader.exec_time_avg_us := 0;
END_IF
stHeader.cycle_exceed_count := nCycleExceedInWnd;
stHeader.rt_violation_count := nRtViolationInWnd;

Tc2_System.MEMSET(ADR(stHeader.task_name), 0, 20);
sTaskName := pTask^.TaskName;
nNameLen := Tc2_Utilities.LEN2(ADR(sTaskName));
IF nNameLen > 20 THEN
    nNameLen := 20;
END_IF
IF nNameLen > 0 THEN
    Tc2_System.MEMCPY(ADR(stHeader.task_name), ADR(sTaskName), nNameLen);
END_IF

(* Copy header to send buffer. *)
Tc2_System.MEMCPY(ADR(abySendBuffer), ADR(stHeader), nHeaderSize);
nOffset := nHeaderSize;

(* Walk the ring from oldest to newest. If we overflowed we want
   chronological order, so start `nRingCount` back from the head. *)
IF nRingCount >= nMaxSamples THEN
    nStartRead := nRingHead; // oldest slot is the one we're about to overwrite
ELSIF nRingCount > nRingHead THEN
    (* Ring wrapped: go back from head by nRingCount, wrapping modulo nMaxSamples. *)
    nStartRead := nMaxSamples - (nRingCount - nRingHead);
ELSE
    nStartRead := nRingHead - nRingCount;
END_IF

FOR nRingIter := 0 TO nRingCount - 1 DO
    nLocalIdx := nStartRead + nRingIter;
    IF nLocalIdx >= nMaxSamples THEN
        nLocalIdx := nLocalIdx - nMaxSamples;
    END_IF
    Tc2_System.MEMCPY(
        ADR(abySendBuffer) + nOffset,
        ADR(aSampleRing[nLocalIdx]),
        nSampleSize
    );
    nOffset := nOffset + nSampleSize;
END_FOR

nBytesToWrite := nOffset;

(* Kick ADSWRITE using the same rising-edge idiom as FB_TcOtelTask:
   reset with WRITE:=FALSE first, then trigger with the full parameter
   set. Subsequent cycles pump the FB with a bare call at the top of
   Call() until BUSY falls. *)
fbAdsWrite(WRITE := FALSE);
fbAdsWrite(
    NETID   := sTcOtelNetId,
    PORT    := nTcOtelPort,
    IDXGRP  := nIdxGroupPushDiag,
    IDXOFFS := nIdxOffsetBatch,
    LEN     := nBytesToWrite,
    SRCADDR := ADR(abySendBuffer),
    WRITE   := TRUE,
    TMOUT   := T#1S
);
bFlushInFlight   := TRUE;
nFlushStartCycle := pTask^.CycleCount;

(* Reset for next window. *)
nRingHead         := 0;
nRingCount        := 0;
nExecTimeMinUs    := 0;
nExecTimeMaxUs    := 0;
nExecTimeSumUs    := 0;
nExecTimeSamples  := 0;
nCycleExceedInWnd := 0;
nRtViolationInWnd := 0;
nCycleCountStart  := 0;
nCycleCountEnd    := 0;
nDcTimeStart      := 0;
nDcTimeEnd        := 0;
bWindowHasSample  := FALSE;
END_METHOD

(*
:Description: Bind this instance to a tc-otel endpoint and its config slot.

Safe to call on every cycle — the first call wires the pointer, further
calls are no-ops. Call from ``PRG_TaskLog.Init`` or during first-cycle
of each task.
*)
METHOD PUBLIC Init : BOOL
VAR_INPUT
    sAmsNetId   : T_AmsNetId;                     // tc-otel AMS net id
    nPort       : UINT;                           // tc-otel ADS port (default 16150)
    pCfg        : REFERENCE TO ST_PushDiagConfig; // per-task config slot
END_VAR
sTcOtelNetId := sAmsNetId;
IF nPort <> 0 THEN
    nTcOtelPort := nPort;
END_IF
pConfig REF= pCfg;
bInitialized := TRUE;
bWindowStartSet := FALSE;
Init := TRUE;
END_METHOD

END_FUNCTION_BLOCK

// ---- POUs/Utils/F_DINT_TO_UINT_MAX.TcPOU
FUNCTION INTERNAL F_DINT_TO_UINT_MAX : UINT
VAR_INPUT
	nValue			: DINT;
	nMaxValue		: UINT;
END_VAR

IF nValue < 0 THEN
	F_DINT_TO_UINT_MAX := 0;
ELSIF nValue > nMaxValue THEN
	F_DINT_TO_UINT_MAX := nMaxValue;
ELSE
	F_DINT_TO_UINT_MAX := DINT_TO_UINT(nValue);
END_IF

END_FUNCTION

// ---- ApiTest.TcPOU
PROGRAM INTERNAL ApiTest
VAR
	nInt			: INT;
	sStr			: STRING;
	fFloat			: REAL;
	fbTrace			: FB_Trace;
	fbSpan			: FB_Span(fbTrace);
END_VAR

// Einfaches Logging
F_Log(E_LogLevel.eInfo, 'Log message')
	.WithLogger('ApiTest')
	.CreateLog();

F_Log(E_LogLevel.eInfo, 'Log Message Arg={structuredArg} Arg={1} Arg=%s')
	.WithTArg(F_StringEx('Arg 1'))
	.WithTArg(F_StringEx('Arg 2'))
	.WithTArg(F_StringEx('Arg 3'))
	.CreateLog();

F_Log(E_LogLevel.eError, 'Log Message Arg={structuredArg} Arg={1} Arg=%s')
	.WithAnyArg(nInt)
	.WithAnyArg(sStr)
	.WithAnyArg(fFloat)
	.CreateLog();

// Einfaches Logging mit expliziten Logger
F_Log(E_LogLevel.eInfo, 'Log Message Arg={structuredArg} Arg={1} Arg=%s')
	.WithLogger('tc-otel.Test')
	.WithTArg(F_StringEx('Arg 1'))
	.WithTArg(F_StringEx('Arg 2'))
	.WithTArg(F_StringEx('Arg 3'))
	.CreateLog();

END_PROGRAM
